RoboDK station: Vertico_Digital_Twin.rdk

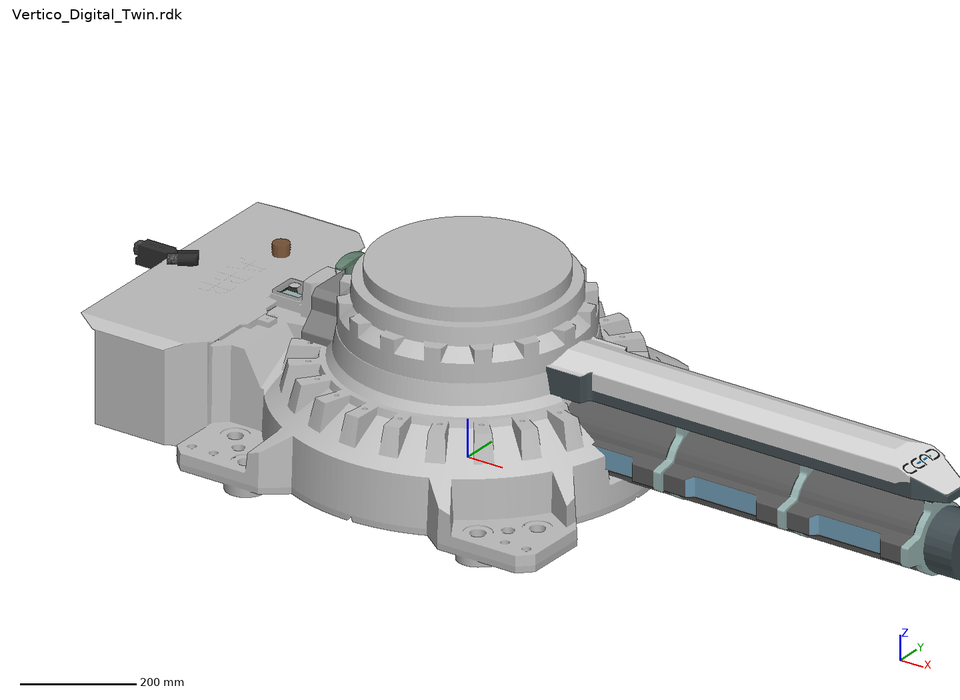
[picture v0: the station drawn from its stored meshes, robots at their saved joint values, targets as dots, program paths as lines]
Station New Station (1) (saved by RoboDK 6.0.4). Poses are relative to the parent item; angles as X-Y-Z fixed-axis rotations.
  - frame ABB IRB 6700-150/3.20 Base at (0, 0, 0) mm
    - robot ABB IRB 6700-150/3.20: 6 axes, payload 150 kg, reach 3200 mm, repeatability 0.06 mm, weight 1280 kg
        joint limits [-170, -65, -180, -300, -130, -360] to [170, 85, 70, 300, 130, 360]; home [0, 0, 0, 0, 0, 0]; saved at [0, 0, 0, 0, 0, 0]
      - tool CEAD Extruder E40, TCP at (1120.5, 0, 123) mm, rotated rx 0 ry 90 rz 0 deg, size 1818.5 x 325.2 x 322 mm
